FUNCTION_BLOCK Process IMPLEMENTS IProcess, I_Station, I_Cyclic, I_Resettable, I_Object
VAR
	_IsClear : BOOL := TRUE;
	_Complete : BOOL;
	_Operating : BOOL;
	_Ready : BOOL := TRUE;
	_Position : LREAL := 0.0;
	_HasMover : BOOL;
	MoverArrive : R_TRIG;
	_MyMover : I_XtsMover;
	_endPos : MC_LREAL;
	_processVelo : MC_LREAL;
	State : INT;
END_VAR

{analysis -2}

METHOD PUBLIC  Cycle : HRESULT
VAR_INPUT
END_VAR
MoverArrive(CLK := _HasMover);
Operation();
IF MoverArrive.Q THEN
	_IsClear := FALSE;
	_Ready := FALSE;
	_Operating := TRUE;
	_Complete := FALSE;
END_IF
END_METHOD

PROPERTY EndPosition : MC_LREAL
GET
EndPosition := _endPos;
END_GET
END_PROPERTY

(*FB_Init is always available implicitly and it is used primarily for initialization.
The return value is not evaluated. For a specific influence, you can also declare the
methods explicitly and provide additional code there with the standard initialization
code. You can evaluate the return value.*)
METHOD FB_Init : BOOL
VAR_INPUT
	(* TRUE: the retain variables are initialized (reset warm / reset cold)*)
	bInitRetains	: BOOL;
	(* TRUE: the instance will be copied to the copy code afterward (online change)   *)
	bInCopyCode	: BOOL;
	Position	: LREAL;
	EndPosition : LREAL;
	ProcessVelocity : LREAL;
END_VAR
_endPos := EndPosition;
_processVelo := ProcessVelocity;
END_METHOD

METHOD HasMover : BOOL
VAR_INPUT
END_VAR
HasMover := _HasMover;
END_METHOD

METHOD IsClear : BOOL
IsClear := _IsClear;
END_METHOD

METHOD isComplete : BOOL
isComplete := _Complete;
END_METHOD

METHOD IsOperating : BOOL
IsOperating := _Operating;
END_METHOD

METHOD IsReady : BOOL
IsReady := _Ready;
END_METHOD

METHOD MyMover : HRESULT
VAR_INPUT
	mover : I_XtsMover;
END_VAR
IF mover = 0 THEN
	MyMover := -1;
	RETURN;
END_IF
_HasMover := TRUE;
_MyMover := mover;
END_METHOD

METHOD PROTECTED Operation : BOOL
CASE State OF
	0:
		IF _Operating THEN
			IF Succeeded(_MyMover.MoveTo(RequiredPosition := _endPos,
							MoveVelocity := _processVelo,
							NonModuloMove := FALSE)) THEN
				State := 1;
			END_IF
		END_IF
	1:
		IF _MyMover.getTrackPosition() = _endPos THEN
			_Operating := FALSE;
			_Complete := TRUE;
			State := 0;
		END_IF
END_CASE	

// IF _Complete AND _HasMover AND_THEN _MyMover.AxisRef.NcToPlc.SetPos > _Position + 50  THEN
// 	_Ready := TRUE;
// 	_HasMover := FALSE;
// 	_IsClear := TRUE;
// 	_MyMover := 0;
// END_IF
END_METHOD

PROPERTY Position : lreal
GET
Position := _Position;
END_GET
END_PROPERTY

PROPERTY ProcessVelocity : MC_LREAL
GET
ProcessVelocity := _processVelo;
END_GET
END_PROPERTY

METHOD RegisterWithParent
VAR_INPUT
	Runner	: I_HostObjects;
END_VAR
Runner.RegisterCyclic(THIS^);
END_METHOD

METHOD Reset : HRESULT
VAR_INPUT
END_VAR
_Complete := FALSE;
_IsClear := TRUE;
_Operating := FALSE;
_Ready := TRUE;
_HasMover := FALSE;
END_METHOD

END_FUNCTION_BLOCK

(* stored: Version 1.1.0.1
   POU Process: Id {5bb3084c-8dc2-4985-92e4-194b505a9bed}, SpecialFunc None
   Folder Status: Id {f15f8ed9-caeb-47bb-9e94-747e6dea9678}
   Method Cycle: Id {898c105c-64a3-42d1-a88c-fca93bd1937e}
   Property EndPosition: Id {7f4a20d7-f0db-4d2e-987f-1dcaac0ba263}
   Get Get: Id {87faf885-3d96-408c-9e10-b4693bedb554}
   Method FB_Init: Id {5e3199be-9a54-4a76-84c3-07069d45f332}
   Method HasMover: Id {1fef3b62-3814-426f-9e0f-bdbf515d1660}
   Method IsClear: Id {aa9c3c67-0da3-4c67-a809-ea7c4fc6f24f}
   Method isComplete: Id {a9fd9f2d-508c-4ae4-8c6d-97dffcefaaa3}
   Method IsOperating: Id {0fd63629-5c93-4ec7-acca-5ba05224e9e4}
   Method IsReady: Id {4549fe33-4b7d-4bec-8cf4-73d1a2e48d3b}
   Method MyMover: Id {d0de5754-d536-4d18-8104-0151b4b47d09}
   Method Operation: Id {4496305a-dcfe-4c87-9747-73150426f565}
   Property Position: Id {27971ba4-3bc4-424c-b956-ef74dcfec010}
   Get Get: Id {1a26a332-bf80-4299-b36a-dae5bd47eff8}
   Property ProcessVelocity: Id {2b95ecf7-a866-474e-93f5-19b6d8e1320a}
   Get Get: Id {25f5b52c-e44e-4bf2-b54e-ddc8a6dd0b98}
   Method RegisterWithParent: Id {329d2fc4-da0f-4271-8758-9b1fd4d1839d}
   Method Reset: Id {34928590-822e-4311-9ea9-b20de4a0cb80} *)
